// LS Electric XG5000 project: LABOLD_CCS
// PLC NewPLC
// module base 0 slot 0: 입력 모듈:XGI-D22A/B (DC 24V 입력, 16점)
// module base 0 slot 1: 출력 모듈:XGQ-TR2A/B (TR 출력, 16점)
// module base 0 slot 2: 아날로그출력 모듈:XGF-DV4A (전압형, 4채널)
// module base 0 slot 3: 아날로그출력 모듈:XGF-DC4A (전류형, 4채널)
// module base 0 slot 4: 아날로그입력 모듈:XGF-AD8A (혼합형, 8채널)
// module base 0 slot 5: EtherNet/IP:XGL-EIPT
// module base 0 slot 6: Cnet:XGL-CH2A

PROGRAM Tag_Test (task: 스캔 프로그램)

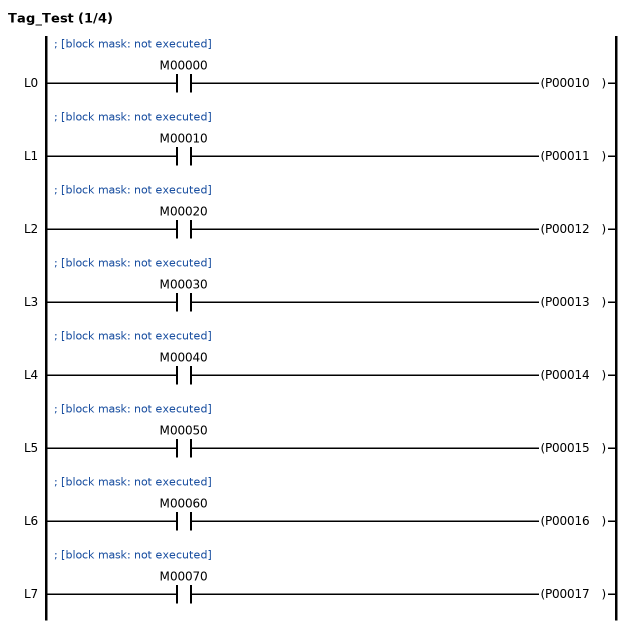
; L0 (block mask: not executed)
LOAD      M00000
OUT       P00010
; L1 (block mask: not executed)
LOAD      M00010
OUT       P00011
; L2 (block mask: not executed)
LOAD      M00020
OUT       P00012
; L3 (block mask: not executed)
LOAD      M00030
OUT       P00013
; L4 (block mask: not executed)
LOAD      M00040
OUT       P00014
; L5 (block mask: not executed)
LOAD      M00050
OUT       P00015
; L6 (block mask: not executed)
LOAD      M00060
OUT       P00016
; L7 (block mask: not executed)
LOAD      M00070
OUT       P00017

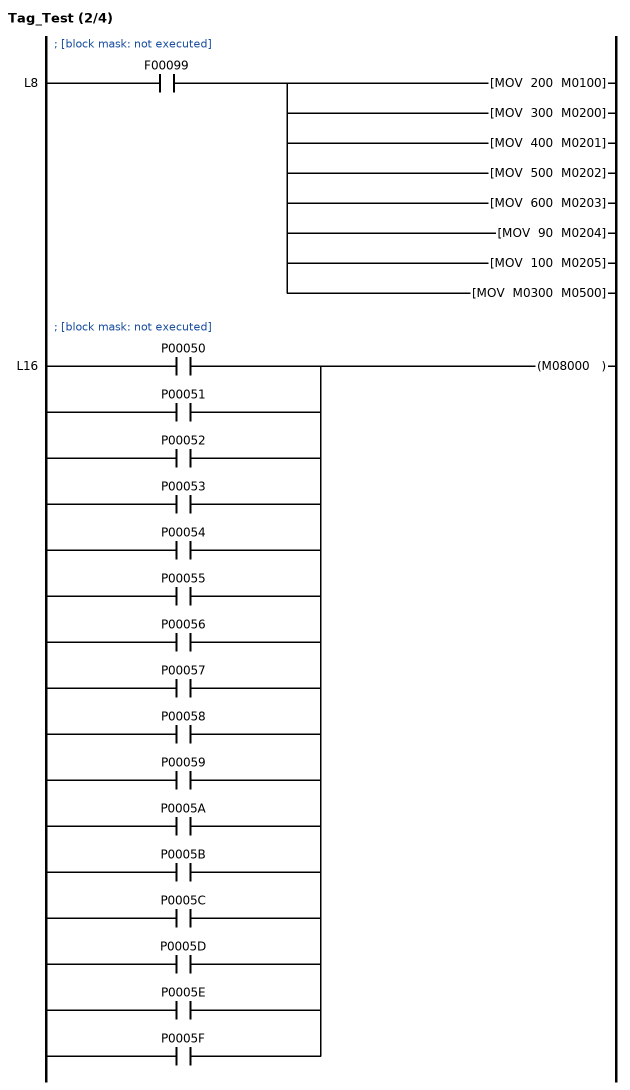
; L8 (block mask: not executed)
LOAD      F00099
MOV       200 M0100
MOV       300 M0200
MOV       400 M0201
MOV       500 M0202
MOV       600 M0203
MOV       90 M0204
MOV       100 M0205
MOV       M0300 M0500
; L16 (block mask: not executed)
LOAD      P00050
OR        P00051
OR        P00052
OR        P00053
OR        P00054
OR        P00055
OR        P00056
OR        P00057
OR        P00058
OR        P00059
OR        P0005A
OR        P0005B
OR        P0005C
OR        P0005D
OR        P0005E
OR        P0005F
OUT       M08000

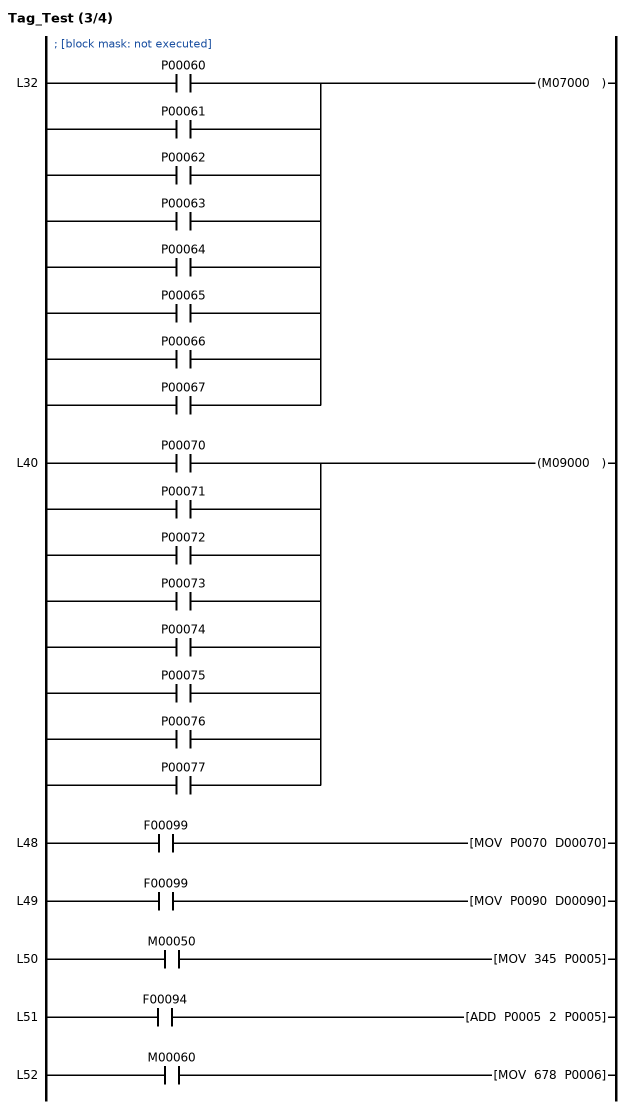
; L32 (block mask: not executed)
LOAD      P00060
OR        P00061
OR        P00062
OR        P00063
OR        P00064
OR        P00065
OR        P00066
OR        P00067
OUT       M07000
; L40
LOAD      P00070
OR        P00071
OR        P00072
OR        P00073
OR        P00074
OR        P00075
OR        P00076
OR        P00077
OUT       M09000
; L48
LOAD      F00099
MOV       P0070 D00070
; L49
LOAD      F00099
MOV       P0090 D00090
; L50
LOAD      M00050
MOV       345 P0005
; L51
LOAD      F00094
ADD       P0005 2 P0005
; L52
LOAD      M00060
MOV       678 P0006

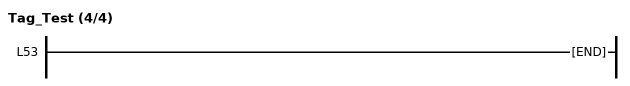
; L53
END

PROGRAM CHECK_SUM_LAYBOLD (task: 스캔 프로그램)
// 레이볼드 터보펌프 컨트롤러의 체크섬 계산하는 방법



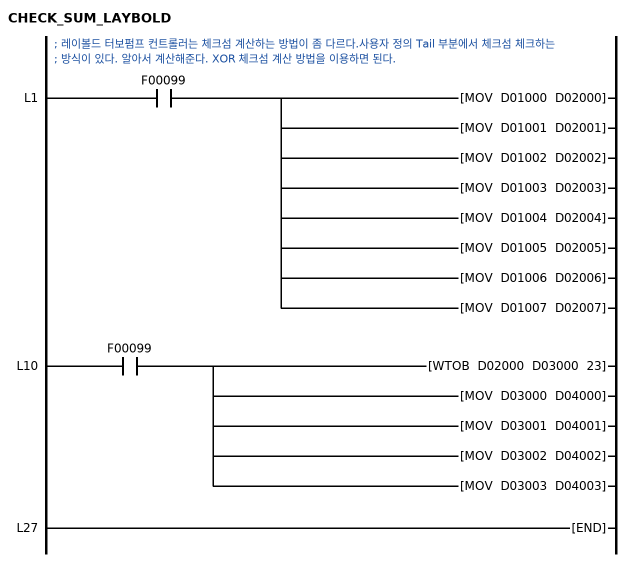
// 레이볼드 터보펌프 컨트롤러는 체크섬 계산하는 방법이 좀 다르다.사용자 정의 Tail 부분에서 체크섬 체크하는 방식이 있다. 알아서 계산해준다. XOR 체크섬 계산 방법을 이용하면 된다.
; L1
LOAD      F00099
MOV       D01000 D02000
MOV       D01001 D02001
MOV       D01002 D02002
MOV       D01003 D02003
MOV       D01004 D02004
MOV       D01005 D02005
MOV       D01006 D02006
MOV       D01007 D02007
; L10
LOAD      F00099
WTOB      D02000 D03000 23
MOV       D03000 D04000
MOV       D03001 D04001
MOV       D03002 D04002
MOV       D03003 D04003
; L27
END